(* PLC project PLC_ForTwinSAFEinTc3, Beckhoff Automation GmbH TwinCAT PLC Control 3.5.0.0 *)
(* stored: creationDateTime 2012-07-11T12:29:45.1632277, modificationDateTime 2012-07-11T12:29:45.1632277 *)

TYPE DUT_ST_InfoDataConnectionIn : STRUCT
  usiMapState : USINT;  (* Safety input connections use this structure *)
  usiMapDiag : USINT;
  byInputSignals : BYTE;
END_STRUCT;
END_TYPE

TYPE DUT_ST_InfoData : STRUCT
  usiMapState : USINT;  (* Safety Groups use this structure *)
  usiMapDiag : USINT;
END_STRUCT;
END_TYPE

TYPE DUT_ST_InfoDataConnectionOut : STRUCT
  usiMapState : USINT;  (* Safety output connections use this structure *)
  usiMapDiag : USINT;
  byOutputSignals : BYTE;
END_STRUCT;
END_TYPE

TYPE DUT_ST_InfoDataFB : STRUCT
  usiMapState : USINT;  (* Safety FBs use this structure *)
  uiMapDiag : UINT;
END_STRUCT;
END_TYPE

TYPE DUT_test : STRUCT
  usiMapState : BYTE;  (* Safety test *)
  uiMapDiag : ARRAY[0..1] OF BYTE;
END_STRUCT;
END_TYPE

TYPE DUT_Test2 : STRUCT
  test_byte : BYTE;
  test_uint : UINT;
END_STRUCT;
END_TYPE

FUNCTION_BLOCK FB_InfoAND
  VAR_INPUT
    stInfoData : DUT_ST_InfoDataFB;
  END_VAR
  VAR_OUTPUT
    sState : STRING;
  END_VAR

                  // AND FB's State
IF stInfoData.usiMapState = 0 THEN
	sState := 'Undefined' ;
	ELSIF stInfoData.usiMapState = 1 THEN
	sState := 'RUN' ;
	ELSIF stInfoData.usiMapState = 2 THEN
	sState := 'STOP' ;
	ELSIF stInfoData.usiMapState = 3 THEN
	sState := 'SAFE' ;
	ELSE
	sState := 'Unknown' ;
END_IF

// The AND FB Has No Diagnostic Byte to Decode
                
END_FUNCTION_BLOCK

FUNCTION_BLOCK FB_InfoConnectionIn
  VAR_INPUT
    stInfoData : DUT_ST_InfoDataConnectionIn;
  END_VAR
  VAR_OUTPUT
    sState : STRING;
    sDiag : STRING;
    xChannel1 : BOOL;
    xChannel2 : BOOL;
    xChannel3 : BOOL;
    xChannel4 : BOOL;
  END_VAR

                  // Safety Terminal's Connection State

// Value 100 (0x64) - The Reset State: The reset state is used to re-initialize 
// the Safety over EtherCAT connection after the power-on or a Safety over EtherCAT 
// communication error
IF stInfoData.usiMapState = 100 THEN
	sState := 'Reset State' ;

// Value 101 (0x65) - The Session State: During the transition to or in the session 
// state a session ID is transferred from the FSoE master to the SFoE slave. which
// in turn responds with its own session ID back to the FSoE master
ELSIF stInfoData.usiMapState = 101 THEN
	sState := 'Session State' ;	

// Value 102 (0x66) - The Connection State: In the connection state a connection ID 
// is transferred from the FSoE master to the FSoE slave
ELSIF stInfoData.usiMapState = 102 THEN
	sState := 'Connection State' ;

// Value 103 (0x67) - The Parameter State: In the parameter state safe communication 
// and device specific application parameters are transferred from the FSoE master 
// to the FSoE slave
ELSIF stInfoData.usiMapState = 103 THEN
	sState := 'Parameter State' ;

// Value 104 (0x68) - The Data Exchange State: In the data state FSoE cycles
// are transferred until either a communications error occurs or an FSoE node
// is stopped locally
ELSIF stInfoData.usiMapState = 104 THEN
	sState := 'Data State' ;

// Value 105 (0x69) - The Shut Down State: In the shut down state the connection 
// was shutdown by one of the communication partners
ELSIF stInfoData.usiMapState = 105 THEN
	sState := 'Shutdown State' ;

// Value is not between 100 and 105 so unknown state which is an error
ELSE
	sState := 'Error' ;
END_IF

// Safety Terminal's Connection Diagnostics

IF stInfoData.usiMapDiag = 0 THEN
	sDiag := 'No Error' ;

// Value		Description
// xxxx 0001	Invalid Command
ELSIF  stInfoData.usiMapDiag.0 = TRUE THEN
	sDiag := 'Invalid Command' ;

// Value		Description
// xxxx 0010	Unknown Command
ELSIF  stInfoData.usiMapDiag.1 = TRUE THEN
	sDiag := 'Unknown Command' ;

// Value		Description
// xxxx 0011	Invalid Connection ID
ELSIF  (stInfoData.usiMapDiag.0 AND stInfoData.usiMapDiag.1) = TRUE THEN
	sDiag := 'Invalid Connection-ID' ;

// Value		Description
// xxxx 0100	Invalid CRC
ELSIF  stInfoData.usiMapDiag.2 = TRUE THEN
	sDiag := 'Invalid CRC' ;

// Value		Description
// xxxx 0101	Watchdog Time Elapsed
ELSIF  (stInfoData.usiMapDiag.0 AND stInfoData.usiMapDiag.2) = TRUE THEN
	sDiag := 'Watchdog Expired' ;
	
// Value		Description
// xxxx 0110	Invalid FSoE Address	
ELSIF  (stInfoData.usiMapDiag.1 AND stInfoData.usiMapDiag.2) = TRUE THEN
	sDiag := 'Invalid FSoE Address' ;

// Value		Description
// xxxx 0111	Invalid Data
ELSIF  (stInfoData.usiMapDiag.0 AND stInfoData.usiMapDiag.1 AND stInfoData.usiMapDiag.2) = TRUE THEN	
	sDiag := 'Invalid Data' ;
	
// Value		Description
// xxxx 1000	Invalid Communication Parameter Length
ELSIF  stInfoData.usiMapDiag.3 = TRUE THEN
	sDiag := 'Invalid Communication Parameter Length' ;

// Value		Description
// xxxx 1001	Invalid Communication Parameters
ELSIF  (stInfoData.usiMapDiag.0 AND stInfoData.usiMapDiag.3) = TRUE THEN
	sDiag := 'Invalid Commuication Parameters' ;

// Value		Description
// xxxx 1010	Invalid User Parameter Length
ELSIF  (stInfoData.usiMapDiag.1 AND stInfoData.usiMapDiag.3) = TRUE THEN
	sDiag := 'Invalid User Parameter Length' ;

// Value		Description
// xxxx 1011	Invalid User PArameters
ELSIF  (stInfoData.usiMapDiag.0 AND stInfoData.usiMapDiag.1 AND stInfoData.usiMapDiag.3) = TRUE THEN	
	sDiag := 'Invalid User Parameters' ;

// Value		Description
// xxxx 1100	FSoE Master Reset	
ELSIF  (stInfoData.usiMapDiag.2 AND stInfoData.usiMapDiag.3) = TRUE THEN
	sDiag := 'FSoE Master Reset' ;

// Value		Description
// 0001 xxxx	FSoE Slave Error Detected
ELSIF  stInfoData.usiMapDiag.4 = TRUE THEN
	sDiag := 'FSoE Slave Error Detected' ;

// Value		Description
// 0010 xxxx	FSoE Slave Reports Failsafe Value Active
ELSIF  stInfoData.usiMapDiag.5 = TRUE THEN
	sDiag := 'FSoE Slave Reports Failsafe Value Active' ;

// Value		Description
// 0100 xxxx	Connection is in Startup
ELSIF  stInfoData.usiMapDiag.6 = TRUE THEN
	sDiag := 'Connection Is In Startup' ;

// Value		Description
// 1000 xxxx	FSoE Master Reports Failsafe Value Active	
ELSIF  stInfoData.usiMapDiag.7 = TRUE THEN
	sDiag := 'FSoE Master Reports Failsafe Value Active' ;	

// Value		Description
// 				Something Not Specifically Annunciated Above.
// 				Maybe a combination of errors are occuring.
ELSE	
	sDiag := 'Error' ;

END_IF


// Safety Terminal's Connection Input Signals
xChannel1 := stInfoData.byInputSignals.0 ;
xChannel2 := stInfoData.byInputSignals.1 ;
xChannel3 := stInfoData.byInputSignals.2 ;
xChannel4 := stInfoData.byInputSignals.3 ;

                
END_FUNCTION_BLOCK

FUNCTION_BLOCK FB_InfoConnectionOut
  VAR_INPUT
    stInfoData : DUT_ST_InfoDataConnectionOut;
  END_VAR
  VAR_OUTPUT
    sState : STRING;
    sDiag : STRING;
    xChannel1 : BOOL;
    xChannel2 : BOOL;
    xChannel3 : BOOL;
    xChannel4 : BOOL;
  END_VAR

                  // Safety Terminal's Connection State

// Value 100 (0x64) - The Reset State: The reset state is used to re-initialize 
// the Safety over EtherCAT connection after the power-on or a Safety over EtherCAT 
// communication error
IF stInfoData.usiMapState = 100 THEN
	sState := 'Reset State' ;

// Value 101 (0x65) - The Session State: During the transition to or in the session 
// state a session ID is transferred from the FSoE master to the SFoE slave. which
// in turn responds with its own session ID back to the FSoE master
ELSIF stInfoData.usiMapState = 101 THEN
	sState := 'Session State' ;	

// Value 102 (0x66) - The Connection State: In the connection state a connection ID 
// is transferred from the FSoE master to the FSoE slave
ELSIF stInfoData.usiMapState = 102 THEN
	sState := 'Connection State' ;

// Value 103 (0x67) - The Parameter State: In the parameter state safe communication 
// and device specific application parameters are transferred from the FSoE master 
// to the FSoE slave
ELSIF stInfoData.usiMapState = 103 THEN
	sState := 'Parameter State' ;

// Value 104 (0x68) - The Data Exchange State: In the data state FSoE cycles
// are transferred until either a communications error occurs or an FSoE node
// is stopped locally
ELSIF stInfoData.usiMapState = 104 THEN
	sState := 'Data State' ;

// Value 105 (0x69) - The Shut Down State: In the shut down state the connection 
// was shutdown by one of the communication partners
ELSIF stInfoData.usiMapState = 105 THEN
	sState := 'Shutdown State' ;

// Value is not between 100 and 105 so unknown state which is an error
ELSE
	sState := 'Error' ;
END_IF

// Safety Terminal's Connection Diagnostics

IF stInfoData.usiMapDiag = 0 THEN
	sDiag := 'No Error' ;

// Value		Description
// xxxx 0001	Invalid Command
ELSIF  stInfoData.usiMapDiag.0 = TRUE THEN
	sDiag := 'Invalid Command' ;

// Value		Description
// xxxx 0010	Unknown Command
ELSIF  stInfoData.usiMapDiag.1 = TRUE THEN
	sDiag := 'Unknown Command' ;

// Value		Description
// xxxx 0011	Invalid Connection ID
ELSIF  (stInfoData.usiMapDiag.0 AND stInfoData.usiMapDiag.1) = TRUE THEN
	sDiag := 'Invalid Connection-ID' ;

// Value		Description
// xxxx 0100	Invalid CRC
ELSIF  stInfoData.usiMapDiag.2 = TRUE THEN
	sDiag := 'Invalid CRC' ;

// Value		Description
// xxxx 0101	Watchdog Time Elapsed
ELSIF  (stInfoData.usiMapDiag.0 AND stInfoData.usiMapDiag.2) = TRUE THEN
	sDiag := 'Watchdog Expired' ;
	
// Value		Description
// xxxx 0110	Invalid FSoE Address	
ELSIF  (stInfoData.usiMapDiag.1 AND stInfoData.usiMapDiag.2) = TRUE THEN
	sDiag := 'Invalid FSoE Address' ;

// Value		Description
// xxxx 0111	Invalid Data
ELSIF  (stInfoData.usiMapDiag.0 AND stInfoData.usiMapDiag.1 AND stInfoData.usiMapDiag.2) = TRUE THEN	
	sDiag := 'Invalid Data' ;
	
// Value		Description
// xxxx 1000	Invalid Communication Parameter Length
ELSIF  stInfoData.usiMapDiag.3 = TRUE THEN
	sDiag := 'Invalid Communication Parameter Length' ;

// Value		Description
// xxxx 1001	Invalid Communication Parameters
ELSIF  (stInfoData.usiMapDiag.0 AND stInfoData.usiMapDiag.3) = TRUE THEN
	sDiag := 'Invalid Commuication Parameters' ;

// Value		Description
// xxxx 1010	Invalid User Parameter Length
ELSIF  (stInfoData.usiMapDiag.1 AND stInfoData.usiMapDiag.3) = TRUE THEN
	sDiag := 'Invalid User Parameter Length' ;

// Value		Description
// xxxx 1011	Invalid User PArameters
ELSIF  (stInfoData.usiMapDiag.0 AND stInfoData.usiMapDiag.1 AND stInfoData.usiMapDiag.3) = TRUE THEN	
	sDiag := 'Invalid User Parameters' ;

// Value		Description
// xxxx 1100	FSoE Master Reset	
ELSIF  (stInfoData.usiMapDiag.2 AND stInfoData.usiMapDiag.3) = TRUE THEN
	sDiag := 'FSoE Master Reset' ;

// Value		Description
// 0001 xxxx	FSoE Slave Error Detected
ELSIF  stInfoData.usiMapDiag.4 = TRUE THEN
	sDiag := 'FSoE Slave Error Detected' ;

// Value		Description
// 0010 xxxx	FSoE Slave Reports Failsafe Value Active
ELSIF  stInfoData.usiMapDiag.5 = TRUE THEN
	sDiag := 'FSoE Slave Reports Failsafe Value Active' ;

// Value		Description
// 0100 xxxx	Connection is in Startup
ELSIF  stInfoData.usiMapDiag.6 = TRUE THEN
	sDiag := 'Connection Is In Startup' ;

// Value		Description
// 1000 xxxx	FSoE Master Reports Failsafe Value Active	
ELSIF  stInfoData.usiMapDiag.7 = TRUE THEN
	sDiag := 'FSoE Master Reports Failsafe Value Active' ;	

// Value		Description
// 				Something Not Specifically Annunciated Above.
// 				Maybe a combination of errors are occuring.
ELSE	
	sDiag := 'Error' ;

END_IF

// Safety Terminal's Connection Output Signals
xChannel1 := stInfoData.byOutputSignals.0 ;
xChannel2 := stInfoData.byOutputSignals.1 ;
xChannel3 := stInfoData.byOutputSignals.2 ;
xChannel4 := stInfoData.byOutputSignals.3 ;

                
END_FUNCTION_BLOCK

FUNCTION_BLOCK FB_InfoConnectionShutdown
  VAR_INPUT
    stInfoData : DUT_ST_InfoDataFB;
  END_VAR
  VAR_OUTPUT
    sState : STRING;
    sDiag : STRING;
  END_VAR

                  // Connection Shutdown FB's State
IF stInfoData.usiMapState = 0 THEN
	sState := 'Undefined' ;
	ELSIF stInfoData.usiMapState = 2 THEN
	sState := 'STOP' ;
	ELSIF stInfoData.usiMapState = 3 THEN
	sState := 'SAFE' ;
	ELSIF stInfoData.usiMapState = 4 THEN
	sState := 'Error' ;
	ELSIF stInfoData.usiMapState = 5 THEN
	sState := 'Reset' ;
	ELSIF stInfoData.usiMapState = 10 THEN
	sState := 'Active' ;
	ELSIF stInfoData.usiMapState = 11 THEN
	sState := 'Deactive' ;
	ELSE
	sState := 'Unknown' ;
END_IF

// Connection Shutdown FB's Diagnostics
IF stInfoData.uiMapDiag = 0 THEN
	sDiag := 'No Error' ;
ELSIF  stInfoData.uiMapDiag = 1 THEN
	sDiag := 'Discrepancy Error Input Group1' ;
ELSE
	sDiag := 'Unknown' ;
END_IF
                
END_FUNCTION_BLOCK

FUNCTION_BLOCK FB_InfoDecoupler
  VAR_INPUT
    stInfoData : DUT_ST_InfoDataFB;
  END_VAR
  VAR_OUTPUT
    sState : STRING;
  END_VAR

                  // Decouple FB's State
IF stInfoData.usiMapState = 0 THEN
	sState := 'Undefined' ;
	ELSIF stInfoData.usiMapState = 1 THEN
	sState := 'RUN' ;
	ELSIF stInfoData.usiMapState = 2 THEN
	sState := 'STOP' ;
ELSE
	sState := 'Unknown' ;
END_IF

// The Decouple FB Has No Diagnostic Byte to Decode
                
END_FUNCTION_BLOCK

FUNCTION_BLOCK FB_InfoEDM
  VAR_INPUT
    stInfoData : DUT_ST_InfoDataFB;
  END_VAR
  VAR_OUTPUT
    sState : STRING;
    sDiag : STRING;
  END_VAR

                  // EDM FB's State
IF stInfoData.usiMapState = 0 THEN
	sState := 'Undefined' ;
	ELSIF stInfoData.usiMapState = 2 THEN
	sState := 'STOP' ;
	ELSIF stInfoData.usiMapState = 4 THEN
	sState := 'ERROR' ;
	ELSIF stInfoData.usiMapState = 5 THEN
	sState := 'RESET' ;
	ELSIF stInfoData.usiMapState = 14 THEN
	sState := 'Monitor-OFF' ;
	ELSIF stInfoData.usiMapState = 15 THEN
	sState := 'Monitor-ON' ;
	ELSE
	sState := 'Unknown' ;
END_IF

// EDM FB's Diagnostics
IF stInfoData.uiMapDiag = 0 THEN
	sDiag := 'No Error' ;
ELSIF  stInfoData.uiMapDiag = 1 THEN
	sDiag := 'Switch-OFF Timer Elapsed' ;
ELSIF  stInfoData.uiMapDiag = 2 THEN
	sDiag := 'Switch-ON Timer Elapsed' ;
ELSE
	sDiag := 'Unknown' ;
END_IF
                
END_FUNCTION_BLOCK

FUNCTION_BLOCK FB_InfoEStop
  VAR_INPUT
    stInfoData : DUT_ST_InfoDataFB;
  END_VAR
  VAR_OUTPUT
    sState : STRING;
    sDiag : STRING;
  END_VAR

                  // EStop FB's State
IF stInfoData.usiMapState = 0 THEN
	sState := 'Undefined' ;
	ELSIF stInfoData.usiMapState = 1 THEN
	sState := 'RUN' ;
	ELSIF stInfoData.usiMapState = 2 THEN
	sState := 'STOP' ;
	ELSIF stInfoData.usiMapState = 3 THEN
	sState := 'SAFE' ;
	ELSIF stInfoData.usiMapState = 4 THEN
	sState := 'ERROR' ;
	ELSIF stInfoData.usiMapState = 5 THEN
	sState := 'RESET' ;
	ELSIF stInfoData.usiMapState = 6 THEN
	sState := 'START' ;
	ELSIF stInfoData.usiMapState = 8 THEN
	sState := 'DELAYOUT' ;
	ELSE
	sState := 'Unknown' ;
END_IF

// EStop FB's Diagnostics
IF stInfoData.uiMapDiag = 0 THEN
	sDiag := 'No Error' ;
	ELSIF stInfoData.uiMapDiag = 1 THEN
	sDiag := 'Discrepancy Error Input Group 1' ;
	ELSIF stInfoData.uiMapDiag = 2 THEN
	sDiag := 'Discrepancy Error Input Group 2' ;
	ELSIF stInfoData.uiMapDiag = 4 THEN
	sDiag := 'Discrepancy Error Input Group 3' ;
	ELSIF stInfoData.uiMapDiag = 8 THEN
	sDiag := 'Discrepancy Error Input Group 4' ;
	ELSIF stInfoData.uiMapDiag = 16 THEN
	sDiag := 'EDM 1 Monitoring Error' ;	
	ELSIF stInfoData.uiMapDiag = 32 THEN
	sDiag := 'EDM 2 Monitoring Error' ;	
	ELSE
	sDiag := 'Unknown' ;
END_IF
                
END_FUNCTION_BLOCK

FUNCTION_BLOCK FB_InfoMON
  VAR_INPUT
    stInfoData : DUT_ST_InfoDataFB;
  END_VAR
  VAR_OUTPUT
    sState : STRING;
    sDiag : STRING;
  END_VAR

                  // Guard Door Monitor FB's State
IF stInfoData.usiMapState = 0 THEN
	sState := 'Undefined' ;
	ELSIF stInfoData.usiMapState = 1 THEN
	sState := 'RUN' ;
	ELSIF stInfoData.usiMapState = 2 THEN
	sState := 'STOP' ;
	ELSIF stInfoData.usiMapState = 3 THEN
	sState := 'SAFE' ;
	ELSIF stInfoData.usiMapState = 4 THEN
	sState := 'ERROR' ;
	ELSIF stInfoData.usiMapState = 5 THEN
	sState := 'RESET' ;
	ELSIF stInfoData.usiMapState = 6 THEN
	sState := 'START' ;
	ELSIF stInfoData.usiMapState = 7 THEN
	sState := 'Error Delay' ;
	ELSIF stInfoData.usiMapState = 8 THEN
	sState := 'DelayOut' ;
	ELSIF stInfoData.usiMapState = 9 THEN
	sState := 'Function Test' ;
	ELSE
	sState := 'Unknown' ;
END_IF

// Guard Door Monitor FB's Diagnostics
IF stInfoData.uiMapDiag = 0 THEN
	sDiag := 'No Error' ;
ELSIF  stInfoData.uiMapDiag = 1 THEN
	sDiag := 'Discrepancy Error of Input Group 1' ;
ELSIF  stInfoData.uiMapDiag = 2 THEN
	sDiag := 'Discrepancy Error of Input Group 2' ;
ELSIF  stInfoData.uiMapDiag = 4 THEN
	sDiag := 'Discrepancy Error of the Secure Inputs' ;
ELSIF  stInfoData.uiMapDiag = 16 THEN
	sDiag := 'EDM 1 Monitoring Error' ;
ELSIF  stInfoData.uiMapDiag = 32 THEN
	sDiag := 'EDM 2 Monitoring Error' ;
ELSE
	sDiag := 'Unknown' ;
END_IF
                
END_FUNCTION_BLOCK

FUNCTION_BLOCK FB_InfoMuting
  VAR_INPUT
    stInfoData : DUT_ST_InfoDataFB;
  END_VAR
  VAR_OUTPUT
    sState : STRING;
    sDiag : STRING;
  END_VAR

                  // Muting FB's State
IF stInfoData.usiMapState = 0 THEN
	sState := 'Undefined' ;
	ELSIF stInfoData.usiMapState = 1 THEN
	sState := 'RUN' ;
	ELSIF stInfoData.usiMapState = 2 THEN
	sState := 'STOP' ;
	ELSIF stInfoData.usiMapState = 3 THEN
	sState := 'SAFE' ;
	ELSIF stInfoData.usiMapState = 4 THEN
	sState := 'ERROR' ;
	ELSIF stInfoData.usiMapState = 5 THEN
	sState := 'RESET' ;
	ELSIF stInfoData.usiMapState = 8 THEN
	sState := 'DelayOut' ;
	ELSIF stInfoData.usiMapState = 9 THEN
	sState := 'Muting 1' ;
	ELSIF stInfoData.usiMapState = 10 THEN
	sState := 'Muting 2' ;
	ELSIF stInfoData.usiMapState = 11 THEN
	sState := 'Muting 3' ;
	ELSIF stInfoData.usiMapState = 12 THEN
	sState := 'Muting 4' ;
	ELSIF stInfoData.usiMapState = 13 THEN
	sState := 'Muting 5' ;
	ELSIF stInfoData.usiMapState = 14 THEN
	sState := 'Muting 6' ;
	ELSIF stInfoData.usiMapState = 15 THEN
	sState := 'Muting 7' ;
	ELSIF stInfoData.usiMapState = 16 THEN
	sState := 'Muting 8' ;
	ELSIF stInfoData.usiMapState = 17 THEN
	sState := 'Muting 9' ;
	ELSE
	sState := 'Unknown' ;
END_IF

// Muting FB's Diagnostics
IF stInfoData.uiMapDiag = 0 THEN
	sDiag := 'No Error' ;
ELSIF  stInfoData.uiMapDiag = 1 THEN
	sDiag := 'Discrepancy Error In Muting Input Group 1' ;
ELSIF  stInfoData.uiMapDiag = 2 THEN
	sDiag := 'Discrepancy Error In OSSD Input Group' ;
ELSIF  stInfoData.uiMapDiag = 4 THEN
	sDiag := 'Discrepancy Error In Muting Input Group 2' ;
ELSIF  stInfoData.uiMapDiag = 16 THEN
	sDiag := 'EDM 1 Monitoring Error' ;
ELSIF  stInfoData.uiMapDiag = 32 THEN
	sDiag := 'EDM 2 Monitoring Error' ;
ELSIF  stInfoData.uiMapDiag = 64 THEN
	sDiag := 'Muting Sequence Was Violated' ;
ELSIF  stInfoData.uiMapDiag = 128 THEN
	sDiag := 'Maximum Muting Time Was Exceeded' ;
ELSE
	sDiag := 'Unknown' ;
END_IF
                
END_FUNCTION_BLOCK

FUNCTION_BLOCK FB_InfoOperationMode
  VAR_INPUT
    stInfoData : DUT_ST_InfoDataFB;
  END_VAR
  VAR_OUTPUT
    sState : STRING;
    sDiag : STRING;
  END_VAR

                  // Operating Mode FB's State
IF stInfoData.usiMapState = 0 THEN
	sState := 'Undefined' ;
	ELSIF stInfoData.usiMapState = 1 THEN
	sState := 'RUN' ;
	ELSIF stInfoData.usiMapState = 2 THEN
	sState := 'STOP' ;
	ELSIF stInfoData.usiMapState = 3 THEN
	sState := 'SAFE' ;
	ELSIF stInfoData.usiMapState = 4 THEN
	sState := 'ERROR' ;
	ELSIF stInfoData.usiMapState = 5 THEN
	sState := 'RESET' ;
	ELSIF stInfoData.usiMapState = 6 THEN
	sState := 'START' ;
	ELSE
	sState := 'Unknown' ;
END_IF

// Operating Mode FB's Diagnostics
IF stInfoData.uiMapDiag = 0 THEN
	sDiag := 'No Error' ;
ELSIF  stInfoData.uiMapDiag = 1 THEN
	sDiag := 'Discrepancy Monitoring Error' ;
ELSE
	sDiag := 'Unknown' ;
END_IF
                
END_FUNCTION_BLOCK

FUNCTION_BLOCK FB_InfoOR
  VAR_INPUT
    stInfoData : DUT_ST_InfoDataFB;
  END_VAR
  VAR_OUTPUT
    sState : STRING;
  END_VAR

                  // OR FB's State
IF stInfoData.usiMapState = 0 THEN
	sState := 'Undefined' ;
	ELSIF stInfoData.usiMapState = 1 THEN
	sState := 'RUN' ;
	ELSIF stInfoData.usiMapState = 2 THEN
	sState := 'STOP' ;
	ELSIF stInfoData.usiMapState = 3 THEN
	sState := 'SAFE' ;
	ELSE
	sState := 'Unknown' ;
END_IF

// The OR FB Has No Diagnostic Byte to Decode
                
END_FUNCTION_BLOCK

FUNCTION_BLOCK FB_InfoRS
  VAR_INPUT
    stInfoData : DUT_ST_InfoDataFB;
  END_VAR
  VAR_OUTPUT
    sState : STRING;
  END_VAR

                  // RS FB's State
IF stInfoData.usiMapState = 0 THEN
	sState := 'Undefined' ;
	ELSIF stInfoData.usiMapState = 2 THEN
	sState := 'STOP' ;
	ELSIF stInfoData.usiMapState = 3 THEN
	sState := 'SAFE' ;
	ELSIF stInfoData.usiMapState = 9 THEN
	sState := 'SET' ;
	ELSE
	sState := 'Unknown' ;
END_IF

// The RS FB Has No Diagnostic Byte to Decode
                
END_FUNCTION_BLOCK

FUNCTION_BLOCK FB_InfoSafetyGroup
  VAR_INPUT
    stInfoData : DUT_ST_InfoData;
  END_VAR
  VAR_OUTPUT
    sState : STRING;
  END_VAR

                  // Safety Group State

// Value 1 - RUN: All function blocks and TwinSAFE connections assigned to the TwinSAFE
// group operate properly, and all TwinSAFE connections assigned to the TwinSAFE 
// group are up and running
IF stInfoData.usiMapState = 1 THEN
	sState := 'RUN - All FBs and Connections Operating Properly' ;

// Value 2 - Stop: The state TwinSAFE goes to after initialization
ELSIF stInfoData.usiMapState = 2 THEN
	sState := 'STOP - State After Initialization' ;

// Value 3 - SAFE: All function blocks and TwinSAFE connections assigned to the TwinSAFE
// group operate properly, and at least one of the TwinSAFE connections
// assigned to the TwinSAFE group is not up and running
ELSIF stInfoData.usiMapState = 3 THEN
	sState := 'SAFE - An Assigned Connection Not Up and Running' ;

// Value 4 - ERROR: At least one assigned function block or one assigned TwinSAFE connection
// has reported an error 
ELSIF stInfoData.usiMapState = 4 THEN
	sState := 'ERROR - FB or Connection in Error State' ;

// Value 5 - RESET: A positive edge (FALSE -> TRUE) for the safety group error Ack
// of a function block or a TwinSAFE connection error was detected on the ERR_ACK input.
// The system is waiting for a negative edge of the ERR_ACK input.
ELSIF stInfoData.usiMapState = 5 THEN
	sState := 'RESET - ErrAck TRUE, Waiting For ErrAck FALSE' ;

// Value 0: Safety group does not exist or safety controller has not been started
ELSE
	sState := 'Unknown' ;
END_IF

// The Safety Group Has No Diagnostic Byte to Decode
                
END_FUNCTION_BLOCK

FUNCTION_BLOCK FB_InfoSR
  VAR_INPUT
    stInfoData : DUT_ST_InfoDataFB;
  END_VAR
  VAR_OUTPUT
    sState : STRING;
  END_VAR

                  // SR FB's State
IF stInfoData.usiMapState = 0 THEN
	sState := 'Undefined' ;
	ELSIF stInfoData.usiMapState = 2 THEN
	sState := 'STOP' ;
	ELSIF stInfoData.usiMapState = 3 THEN
	sState := 'SAFE' ;
	ELSIF stInfoData.usiMapState = 9 THEN
	sState := 'SET' ;
	ELSE
	sState := 'Unknown' ;
END_IF

// The SR FB Has No Diagnostic Byte to Decode
                
END_FUNCTION_BLOCK

FUNCTION_BLOCK FB_InfoTOF
  VAR_INPUT
    stInfoData : DUT_ST_InfoDataFB;
  END_VAR
  VAR_OUTPUT
    sState : STRING;
  END_VAR

                  // Timer-OFF (TOF) FB's State
IF stInfoData.usiMapState = 0 THEN
	sState := 'Undefined' ;
	ELSIF stInfoData.usiMapState = 1 THEN
	sState := 'RUN' ;
	ELSIF stInfoData.usiMapState = 2 THEN
	sState := 'STOP' ;
	ELSIF stInfoData.usiMapState = 3 THEN
	sState := 'SAFE' ;
	ELSIF stInfoData.usiMapState = 8 THEN
	sState := 'DelayOut' ;
	ELSE
	sState := 'Unknown' ;
END_IF

// The Timer-OFF (TOF) FB Has No Diagnostic Byte to Decode
                
END_FUNCTION_BLOCK

FUNCTION_BLOCK FB_InfoTON
  VAR_INPUT
    stInfoData : DUT_ST_InfoDataFB;
  END_VAR
  VAR_OUTPUT
    sState : STRING;
  END_VAR

                  // Timer-ON (TON) FB's State
IF stInfoData.usiMapState = 0 THEN
	sState := 'Undefined' ;
	ELSIF stInfoData.usiMapState = 1 THEN
	sState := 'RUN' ;
	ELSIF stInfoData.usiMapState = 2 THEN
	sState := 'STOP' ;
	ELSIF stInfoData.usiMapState = 3 THEN
	sState := 'SAFE' ;
	ELSIF stInfoData.usiMapState = 9 THEN
	sState := 'DelayIn' ;
	ELSE
	sState := 'Unknown' ;
END_IF

// The Timer-ON (TON) FB Has No Diagnostic Byte to Decode
                
END_FUNCTION_BLOCK

FUNCTION_BLOCK FB_InfoTwoHand
  VAR_INPUT
    stInfoData : DUT_ST_InfoDataFB;
  END_VAR
  VAR_OUTPUT
    sState : STRING;
    sDiag : STRING;
  END_VAR

                  // Two-Hand Tie Down FB's State
IF stInfoData.usiMapState = 0 THEN
	sState := 'Undefined' ;
	ELSIF stInfoData.usiMapState = 1 THEN
	sState := 'RUN' ;
	ELSIF stInfoData.usiMapState = 2 THEN
	sState := 'STOP' ;
	ELSIF stInfoData.usiMapState = 3 THEN
	sState := 'SAFE' ;
	ELSIF stInfoData.usiMapState = 4 THEN
	sState := 'ERROR' ;
	ELSIF stInfoData.usiMapState = 5 THEN
	sState := 'RESET' ;
	ELSIF stInfoData.usiMapState = 6 THEN
	sState := 'START' ;
	ELSIF stInfoData.usiMapState = 11 THEN
	sState := '1BUTTON' ;
	ELSIF stInfoData.usiMapState = 12 THEN
	sState := '2BUTTON' ;
	ELSIF stInfoData.usiMapState = 13 THEN
	sState := 'RELEASE' ;
	ELSE
	sState := 'Unknown' ;
END_IF

// Two-Hand Tie Down FB's Diagnostics
IF stInfoData.uiMapDiag = 0 THEN
	sDiag := 'No Error' ;
	ELSIF stInfoData.uiMapDiag = 1 THEN
	sDiag := 'Discrepancy Error Input Group 1' ;
	ELSIF stInfoData.uiMapDiag = 2 THEN
	sDiag := 'Discrepancy Error Input Group 2' ;
	ELSIF stInfoData.uiMapDiag = 4 THEN
	sDiag := 'Discrepancy Error Between Input Groups' ;
	ELSE
	sDiag := 'Unknown' ;
END_IF
                
END_FUNCTION_BLOCK

FUNCTION_BLOCK FB_PleaseExplain
  VAR_INPUT
    stInfoData : DUT_test2;
  END_VAR
  VAR_OUTPUT
    sState : STRING;
  END_VAR

                   // does nothing but look at the data size of DUT_Test2
 ;
                
END_FUNCTION_BLOCK

PROGRAM MAIN
  VAR
    fb_InfoSafetyGroup1 : FB_InfoSafetyGroup;
    fb_InfoConnection1 : FB_InfoConnectionIn;
    fb_InfoConnection2 : FB_InfoConnectionOut;
    fb_InfoAND : FB_InfoAND;
    fb_InfoEStop : FB_InfoEStop;
    fb_InfoAND2 : FB_InfoAND;
    fb_InfoTON : FB_InfoTON;
    fb_InfoTOF : FB_InfoTOF;
    fb_InfoEDM : FB_InfoEDM;
  END_VAR

                  // Most Important Safety Project Info!!!
q_udiHMI_SerialNumber := g_udiTS_SerialNumber ;
q_uiHMI_ProjectCRC := g_uiTS_ProjectCRC ;

// Commands to TwinSAFE controller's safety  group
g_xTS_ErrAck := q_xHMI_ErrAckPB ;
g_xTS_EStop_Reset := q_xHMI_EStopResetPB ;

// Feedback from TwinSAFE controller's safety group
q_xHMI_FBerrorLT := g_xTS_FBerror ;
q_xHMI_COMerrorLT := g_xTS_COMerror ;

// Feedback from TwinSAFE controller's Function Blocks
q_xHMI_EDMerrorLT := g_xTS_EDM_Error ;
q_xHMI_EStop_CompleteLT := g_xTS_EStop_Complete ;
q_xHMI_EStop_errorLT := g_xTS_EStop_Error ;
q_xHMI_EStop_OFF_Delay_CompleteLT := g_xTS_EStop_OFF_Delay_Complete ;
q_xHMI_EStop_ON_Delay_CompleteLT := g_xTS_EStop_ON_Delay_Complete ;

// TwinSAFE Group 1 Info
fb_InfoSafetyGroup1(
						stInfoData:= 	g_stTS_InfoGroup1, 
						sState=> 		g_sHMI_StatusGroup1 );

// TwinSAFE Connection 1 Info to EL1904 safety terminal
fb_InfoConnection1(
						stInfoData:= 	g_stTS_InfoConnection1, 
						sState=> 		g_sHMI_StateConn1, 
						sDiag=> 		g_sHMI_DiagConn1, 
						xChannel1=> 	g_xHMI_EL1904Ch1, 
						xChannel2=> 	g_xHMI_EL1904Ch2, 
						xChannel3=> 	g_xHMI_EL1904Ch3, 
						xChannel4=> 	g_xHMI_EL1904Ch4 );
	
// TwinSAFE Connection 2 Info to EL2904 safety terminal
fb_InfoConnection2(
						stInfoData:= 	g_stTS_InfoConnection2, 
						sState=> 		g_sHMI_StateConn2, 
						sDiag=> 		g_sHMI_DiagConn2, 
						xChannel1=> 	g_xHMI_EL2904Ch1, 
						xChannel2=> 	g_xHMI_EL2904Ch2, 
						xChannel3=> 	g_xHMI_EL2904Ch3, 
						xChannel4=> 	g_xHMI_EL2904Ch4 );	
								
// TwinSAFE First AND safety FB Info
fb_InfoAND(				stInfoData:= 	g_stTS_InfoAND1, 
						sState=> 		g_sHMI_StatusAND1 );

// TwinSAFE ESTOP safety FB Info
fb_InfoEStop(			stInfoData:= 	g_stTS_InfoEStop1, 
						sState=> 		g_sHMI_StatusEStop1, 		
						sDiag=> 		g_sHMI_DiagEStop1 );

// TwinSAFE Second AND safety FB Info
fb_InfoAND2(			stInfoData:= 	g_stTS_InfoAND2, 
						sState=> 		g_sHMI_StatusAND2 );
						
// TwinSAFE TON safety FB Info
fb_InfoTON(				stInfoData:= 	g_stTS_InfoTON, 
						sState=> 		g_sHMI_StatusTON );

// TwinSAFE TOF safety FB Info
fb_InfoTOF(				stInfoData:= 	g_stTS_InfoTOF, 
						sState=> 		g_sHMI_StatusTOF );

// TwinSAFE EDM safety FB Info
fb_InfoEDM(				stInfoData:= 	g_stTS_InfoEDM, 
						sState=> 		g_sHMI_StatusEDM, 
						sDiag=> 		g_sHMI_DiagEDM );						

// st_test.test_byte := fb_InfoAND.stInfoData.usiMapState;
// MEMCPY(ADR(st_test.test_uint) , ADR(fb_InfoAND.stInfoData.uiMapDiag) , n:=SIZEOF(fb_InfoAND.stInfoData.uiMapDiag) );
						
//fb_PleaseExplain(		stInfoData:= g_stTS_InfoFromAnyFB, 
//						sState=> 							);

                
END_PROGRAM

CONFIGURATION Application
  RESOURCE PLC_ForTwinSAFEinTc3 ON PLC
    VAR_GLOBAL  (* TC_GLOBAL_IID_LIST *)
      {attribute 'tc_no_symbol'}
      IID_ITcUnknown : IID := (Data1 := 16#1, Data2 := 16#0, Data3 := 16#0, Data4 := [16#E0, 16#0, 16#0, 16#0, 16#0, 16#0, 16#0, 16#64]);  (* Interface ID for interface ITcUnknown *)
      {attribute 'tc_no_symbol'}
      IID_ITComObjCon : IID := (Data1 := 16#16, Data2 := 16#0, Data3 := 16#0, Data4 := [16#E0, 16#0, 16#0, 16#0, 16#0, 16#0, 16#0, 16#64]);  (* Interface ID for interface ITComObjCon *)
      {attribute 'tc_no_symbol'}
      IID_ITComObjRes : IID := (Data1 := 16#14, Data2 := 16#0, Data3 := 16#0, Data4 := [16#E0, 16#0, 16#0, 16#0, 16#0, 16#0, 16#0, 16#64]);  (* Interface ID for interface ITComObjRes *)
      {attribute 'tc_no_symbol'}
      IID_ITComObjInd : IID := (Data1 := 16#13, Data2 := 16#0, Data3 := 16#0, Data4 := [16#E0, 16#0, 16#0, 16#0, 16#0, 16#0, 16#0, 16#64]);  (* Interface ID for interface ITComObjInd *)
      {attribute 'tc_no_symbol'}
      IID_ITcBaseClassFactory : IID := (Data1 := 16#18, Data2 := 16#0, Data3 := 16#0, Data4 := [16#E0, 16#0, 16#0, 16#0, 16#0, 16#0, 16#0, 16#64]);  (* Interface ID for interface ITcBaseClassFactory *)
      {attribute 'tc_no_symbol'}
      IID_ITComObjectServer : IID := (Data1 := 16#30, Data2 := 16#0, Data3 := 16#0, Data4 := [16#E0, 16#0, 16#0, 16#0, 16#0, 16#0, 16#0, 16#64]);  (* Interface ID for interface ITComObjectServer *)
      {attribute 'tc_no_symbol'}
      IID_ITcTask : IID := (Data1 := 16#2000002, Data2 := 16#0, Data3 := 16#0, Data4 := [16#E0, 16#0, 16#0, 16#0, 16#0, 16#0, 16#0, 16#64]);  (* Interface ID for interface ITcTask *)
      {attribute 'tc_no_symbol'}
      IID_ITcCyclic : IID := (Data1 := 16#3000010, Data2 := 16#0, Data3 := 16#0, Data4 := [16#E0, 16#0, 16#0, 16#0, 16#0, 16#0, 16#0, 16#64]);  (* Interface ID for interface ITcCyclic *)
      {attribute 'tc_no_symbol'}
      IID_ITcPostCyclic : IID := (Data1 := 16#3000025, Data2 := 16#0, Data3 := 16#0, Data4 := [16#E0, 16#0, 16#0, 16#0, 16#0, 16#0, 16#0, 16#64]);  (* Interface ID for interface ITcPostCyclic *)
      {attribute 'tc_no_symbol'}
      IID_ITcIoCyclic : IID := (Data1 := 16#3000011, Data2 := 16#0, Data3 := 16#0, Data4 := [16#E0, 16#0, 16#0, 16#0, 16#0, 16#0, 16#0, 16#64]);  (* Interface ID for interface ITcIoCyclic *)
      {attribute 'tc_no_symbol'}
      IID_ITcPersist : IID := (Data1 := 16#2, Data2 := 16#0, Data3 := 16#0, Data4 := [16#E0, 16#0, 16#0, 16#0, 16#0, 16#0, 16#0, 16#64]);  (* Interface ID for interface ITcPersist *)
      {attribute 'tc_no_symbol'}
      IID_ITComCreateInstance : IID := (Data1 := 16#31, Data2 := 16#0, Data3 := 16#0, Data4 := [16#E0, 16#0, 16#0, 16#0, 16#0, 16#0, 16#0, 16#64]);  (* Interface ID for interface ITComCreateInstance *)
      {attribute 'tc_no_symbol'}
      IID_ITComObject : IID := (Data1 := 16#12, Data2 := 16#0, Data3 := 16#0, Data4 := [16#E0, 16#0, 16#0, 16#0, 16#0, 16#0, 16#0, 16#64]);  (* Interface ID for interface ITComObject *)
      {attribute 'tc_no_symbol'}
      IID_ITComObjReq : IID := (Data1 := 16#15, Data2 := 16#0, Data3 := 16#0, Data4 := [16#E0, 16#0, 16#0, 16#0, 16#0, 16#0, 16#0, 16#64]);  (* Interface ID for interface ITComObjReq *)
      {attribute 'tc_no_symbol'}
      IID_ITcRTimeTask : IID := (Data1 := 16#2000003, Data2 := 16#0, Data3 := 16#0, Data4 := [16#E0, 16#0, 16#0, 16#0, 16#0, 16#0, 16#0, 16#64]);  (* Interface ID for interface ITcRTimeTask *)
      {attribute 'tc_no_symbol'}
      IID_ITcRTime : IID := (Data1 := 16#200000D, Data2 := 16#0, Data3 := 16#0, Data4 := [16#E0, 16#0, 16#0, 16#0, 16#0, 16#0, 16#0, 16#64]);  (* Interface ID for interface ITcRTime *)
      {attribute 'tc_no_symbol'}
      IID_ITcPreInputCyclic : IID := (Data1 := 16#3000017, Data2 := 16#0, Data3 := 16#0, Data4 := [16#E0, 16#0, 16#0, 16#0, 16#0, 16#0, 16#0, 16#64]);  (* Interface ID for interface ITcPreInputCyclic *)
      {attribute 'tc_no_symbol'}
      IID_ITcWatchSource : IID := (Data1 := 16#3000018, Data2 := 16#0, Data3 := 16#0, Data4 := [16#E0, 16#0, 16#0, 16#0, 16#0, 16#0, 16#0, 16#64]);  (* Interface ID for interface ITcWatchSource *)
      {attribute 'tc_no_symbol'}
      IID_ITcCyclicCaller : IID := (Data1 := 16#300001E, Data2 := 16#0, Data3 := 16#0, Data4 := [16#E0, 16#0, 16#0, 16#0, 16#0, 16#0, 16#0, 16#64]);  (* Interface ID for interface ITcCyclicCaller *)
      {attribute 'tc_no_symbol'}
      IID_ITcPostCyclicCaller : IID := (Data1 := 16#3000026, Data2 := 16#0, Data3 := 16#0, Data4 := [16#E0, 16#0, 16#0, 16#0, 16#0, 16#0, 16#0, 16#64]);  (* Interface ID for interface ITcPostCyclicCaller *)
      {attribute 'tc_no_symbol'}
      IID_ITcIoCyclicCaller : IID := (Data1 := 16#300001F, Data2 := 16#0, Data3 := 16#0, Data4 := [16#E0, 16#0, 16#0, 16#0, 16#0, 16#0, 16#0, 16#64]);  (* Interface ID for interface ITcIoCyclicCaller *)
      {attribute 'tc_no_symbol'}
      IID_ITcADI : IID := (Data1 := 16#3000012, Data2 := 16#0, Data3 := 16#0, Data4 := [16#E0, 16#0, 16#0, 16#0, 16#0, 16#0, 16#0, 16#64]);  (* Interface ID for interface ITcADI *)
      {attribute 'tc_no_symbol'}
      IID_ITComLicenseServer : IID := (Data1 := 16#1010000, Data2 := 16#0, Data3 := 16#0, Data4 := [16#E0, 16#0, 16#0, 16#0, 16#0, 16#0, 16#0, 16#64]);  (* Interface ID for interface ITComLicenseServer *)
      {attribute 'tc_no_symbol'}
      IID_ITcAppServices : IID := (Data1 := 16#8500102, Data2 := 16#0, Data3 := 16#0, Data4 := [16#E0, 16#0, 16#0, 16#0, 16#0, 16#0, 16#0, 16#64]);  (* Interface ID for interface ITcAppServices *)
      {attribute 'tc_no_symbol'}
      IID_ITcAppServices2 : IID := (Data1 := 16#8500104, Data2 := 16#0, Data3 := 16#0, Data4 := [16#E0, 16#0, 16#0, 16#0, 16#0, 16#0, 16#0, 16#64]);  (* Interface ID for interface ITcAppServices2 *)
      {attribute 'tc_no_symbol'}
      IID_ITcNcDcConvert : IID := (Data1 := 16#5000005, Data2 := 16#0, Data3 := 16#0, Data4 := [16#E0, 16#0, 16#0, 16#0, 16#0, 16#0, 16#0, 16#64]);  (* Interface ID for interface ITcNcDcConvert *)
      {attribute 'tc_no_symbol'}
      IID_ITcNcDcConvert2 : IID := (Data1 := 16#5000006, Data2 := 16#0, Data3 := 16#0, Data4 := [16#E0, 16#0, 16#0, 16#0, 16#0, 16#0, 16#0, 16#64]);  (* Interface ID for interface ITcNcDcConvert2 *)
    END_VAR
    VAR_GLOBAL  (* GVL_TwinSAFE *)
      g_uiTS_ProjectCRC AT %I* : UINT;  (* TwinSAFE project CRC *)
      q_uiHMI_ProjectCRC : UINT;
      g_udiTS_SerialNumber AT %I* : UDINT;
      q_udiHMI_SerialNumber : UDINT;
      g_xTS_ErrAck AT %Q* : BOOL;  (* Commands to TwinSAFE controller's safety group *)
      q_xHMI_ErrAckPB : BOOL;
      g_xTS_EStop_Reset AT %Q* : BOOL;
      q_xHMI_EStopResetPB : BOOL;
      g_xTS_FBerror AT %I* : BOOL;  (* Feedback from TwinSAFE controller's safety group *)
      q_xHMI_FBerrorLT : BOOL;
      g_xTS_COMerror AT %I* : BOOL;
      q_xHMI_COMerrorLT : BOOL;
      g_xTS_EDM_Error AT %I* : BOOL;  (* Feedback from TwinSAFE controller's Function Blocks *)
      q_xHMI_EDMerrorLT : BOOL;
      g_xTS_EStop_Complete AT %I* : BOOL;
      q_xHMI_EStop_CompleteLT : BOOL;
      g_xTS_EStop_Error AT %I* : BOOL;
      q_xHMI_EStop_errorLT : BOOL;
      g_xTS_EStop_OFF_Delay_Complete AT %I* : BOOL;
      q_xHMI_EStop_OFF_Delay_CompleteLT : BOOL;
      g_xTS_EStop_ON_Delay_Complete AT %I* : BOOL;
      q_xHMI_EStop_ON_Delay_CompleteLT : BOOL;
      g_stTS_InfoGroup1 AT %I* : DUT_ST_InfoData;  (* Safety Group1 Info *)
      g_sHMI_StatusGroup1 : STRING;
      g_stTS_InfoConnection1 AT %I* : DUT_ST_InfoDataConnectionIn;  (* Safety Connection1 Info *)
      g_sHMI_StateConn1 : STRING;
      g_sHMI_DiagConn1 : STRING;
      g_xHMI_EL1904Ch1 : BOOL;
      g_xHMI_EL1904Ch2 : BOOL;
      g_xHMI_EL1904Ch3 : BOOL;
      g_xHMI_EL1904Ch4 : BOOL;
      g_stTS_InfoConnection2 AT %I* : DUT_ST_InfoDataConnectionOut;  (* Safety Connection2 Info *)
      g_sHMI_StateConn2 : STRING;
      g_sHMI_DiagConn2 : STRING;
      g_xHMI_EL2904Ch1 : BOOL;
      g_xHMI_EL2904Ch2 : BOOL;
      g_xHMI_EL2904Ch3 : BOOL;
      g_xHMI_EL2904Ch4 : BOOL;
      g_stTS_InfoAND1 AT %I* : DUT_ST_InfoDataFB;  (* Safety AND#1 FB Info *)
      g_sHMI_StatusAND1 : STRING;
      g_stTS_InfoEStop1 AT %I* : DUT_ST_InfoDataFB;  (* Safety EStop#1 FB Info *)
      g_sHMI_StatusEStop1 : STRING;
      g_sHMI_DiagEStop1 : STRING;
      g_stTS_InfoAND2 AT %I* : DUT_ST_InfoDataFB;  (* Safety AND#2 FB Info *)
      g_sHMI_StatusAND2 : STRING;
      g_stTS_InfoTON AT %I* : DUT_ST_InfoDataFB;  (* Safety TON FB Info *)
      g_sHMI_StatusTON : STRING;
      g_stTS_InfoTOF AT %I* : DUT_ST_InfoDataFB;  (* Safety TOF FB Info *)
      g_sHMI_StatusTOF : STRING;
      g_stTS_InfoEDM AT %I* : DUT_ST_InfoDataFB;  (* Safety EDM FB Info *)
      g_sHMI_StatusEDM : STRING;
      g_sHMI_DiagEDM : STRING;
    END_VAR
    TASK PlcTask(INTERVAL := T#10ms, PRIORITY := 20);
    PROGRAM MAIN WITH PlcTask : MAIN;
  END_RESOURCE
END_CONFIGURATION
